{attribute 'qualified_only'}
{attribute 'strict'}
{attribute 'to_string'}
TYPE E_AXIS_CTRL :
(
  AXIS_NULL,   // null command
  AXIS_INIT,
  AXIS_DISABLE,
  AXIS_ENABLE,

  AXIS_IDLE     := 10, // clear axis and enable
  AXIS_HOME,
  AXIS_MOVE_POS,
  AXIS_MOVE_VELO,
  AXIS_HALT,
  AXIS_STOP,
  AXIS_SEND_TO_POS,

  AXIS_RESET              := 19,
  AXIS_STARTUP            := 20,

  AXIS_MOVE_BUFFER        := 30,
  AXIS_MOVE_BUFFER_VELO,

  AXIS_PARAMETER_READ     := 40, // command for reading and writing parameter
  AXIS_PARAMETER_WRITE,
  AXIS_PARAMETER_WRITE_PERSISTENT,


  AXIS_GEAR_IN            := 50,
  AXIS_GEAR_OUT,
  AXIS_GEAR_IN_MULTIMASTER,

  CAM_INIT                := 60,
  CAM_IN,
  CAM_OUT,
  CAM_SCALING,
  CAM_INFO,
  CAM_RD_MOTION_FUNCTION,
  CAM_RD_MOTION_FUNCTION_POINT,
  CAM_RD_MOTION_FUNCTIONS_VALUES,
  CAM_WRT_MOTION_FUNCTION,
  CAM_WRT_MOTION_FUNCTION_POINT,

  FLY_GEAR_IN_POS         := 70,
  FLY_GEAR_IN_VELO

)UINT;
END_TYPE

(* stored: Version 1.1.0.1, ProductVersion 3.1.4026.18
   DUT E_AXIS_CTRL: Id {784d8a43-f813-0ae6-1900-42616ecae467} *)
